FUNCTION_BLOCK FB_Controller_PI EXTENDS FB_Controller_P
VAR_INPUT
END_VAR
VAR_OUTPUT
END_VAR
VAR
	_Tn	: TIME;
END_VAR

// Executes the controller and returns the control output.
METHOD Execute
VAR_OUTPUT
	controllerOutput	: LREAL;	// Controller result
END_VAR
PID.fTn := SUPER^.TimeToSeconds(_Tn);
SUPER^.Execute();
END_METHOD

// Gets or sets the integration action time.
PROPERTY Tn : TIME
GET
Tn := _Tn;
END_GET
SET
_Tn := Tn;
END_SET
END_PROPERTY

END_FUNCTION_BLOCK

(* stored: Version 1.1.0.1, ProductVersion 3.1.4024.15
   POU FB_Controller_PI: Id {cebf8388-c6b7-0e55-16da-d4e5b20ae531}, SpecialFunc None
   Method Execute: Id {27e74276-09b5-04b2-31da-a99e5e710905}
   Property Tn: Id {42266395-9c97-0108-2576-85c5a3ee3fe3}
   Get Get: Id {795daa74-731f-07c9-2bfd-ce189beb5f0c}
   Set Set: Id {ff590ad5-0d15-02ce-146d-3154f4d8b6d1} *)
